// TwinCAT 3 PLC project ReleaseManager
// ProgramVersion: 3.1.4023.0
// libraries:
//   Tc2_Standard, * (Beckhoff Automation GmbH)
//   Tc2_System, * (Beckhoff Automation GmbH)
//   Tc3_Module, * (Beckhoff Automation GmbH)
// project tree:
//   / PlcTask.TcTTO
//   POUs/ MAIN.TcPOU, ReleaseClient.TcPOU, ReleaseHybrid.TcPOU, ReleaseMaster.TcPOU, TestModule_1.TcPOU, TestModule_2.TcPOU, TestModule_3.TcPOU
// real-time tasks:
//   TASK PlcTask: cycle T#10ms, priority 20, ADS port 350

CONFIGURATION ReleaseManager
    RESOURCE PLC ON TwinCAT3
        TASK PlcTask(INTERVAL := T#10ms, PRIORITY := 20);
        PROGRAM MAIN WITH PlcTask : MAIN;
    END_RESOURCE
END_CONFIGURATION

// ---- POUs/MAIN.TcPOU
PROGRAM MAIN
VAR
	fbTestModule1 : TestModule_1;
	fbTestModule2 : TestModule_2;
	fbTestModule3,fbTestModule4,fbTestModule5 : TestModule_3;
END_VAR

fbTestModule1();
fbTestModule2();

//fbTestModule1.fbNextStationReleaseClient.bReleasePresent := fbTestModule2.fbNextStationReleaseMaster.bSetRelease;
//fbTestModule2.fbNextStationReleaseMaster.bReleaseAckIn := fbTestModule1.fbNextStationReleaseClient.bReleaseAckOut;

fbTestModule2.fbNextStationReleaseMaster.SetReleaseClient(fbTestModule1.fbNextStationReleaseClient);
fbTestModule3.fbNextStationReleaseHybrid.SetReleaseClient(fbTestModule4.fbNextStationReleaseHybrid);
fbTestModule4.fbNextStationReleaseHybrid.SetReleaseClient(fbTestModule5.fbNextStationReleaseHybrid);

END_PROGRAM

// ---- POUs/TestModule_1.TcPOU
FUNCTION_BLOCK TestModule_1
VAR_INPUT
	fbNextStationReleaseClient : ReleaseClient;
END_VAR
VAR_OUTPUT
END_VAR
VAR
END_VAR

fbNextStationReleaseClient();

END_FUNCTION_BLOCK

// ---- POUs/ReleaseClient.TcPOU
FUNCTION_BLOCK ReleaseClient
VAR_INPUT
	bReleasePresent : BOOL;
END_VAR

VAR_OUTPUT
	bReleaseAckOut : BOOL;
	bLastHandshakeSuccesful : BOOL;
	bMasterAbortedLastHandshake : BOOL;
END_VAR

VAR
	fbReleasePresentEvent : R_TRIG;
	fbReleaseGoneEvent : F_TRIG;
	fbReleaseAckOutEvent : R_TRIG;
	fbReleaseAckOutGoneEvent : F_TRIG;
END_VAR

fbReleasePresentEvent(CLK:=bReleasePresent);
fbReleaseAckOutEvent(CLK:=bReleaseAckOut);
fbReleaseGoneEvent(CLK:=bReleasePresent);
fbReleaseAckOutGoneEvent(CLK:=bReleaseAckOut);

IF fbReleaseAckOutEvent.Q
THEN
	OnReleaseAckOut();
END_IF

IF fbReleasePresentEvent.Q
THEN
	OnReleasePresent();
END_IF

IF fbReleaseGoneEvent.Q
THEN
	OnReleaseGone();
END_IF

IF fbReleaseAckOutGoneEvent.Q
THEN
	OnHandshakeSuccessful();
END_IF

METHOD OnHandshakeSuccessful : BOOL
VAR_INPUT
END_VAR
bLastHandshakeSuccesful := TRUE;
END_METHOD

METHOD OnReleaseAckOut : BOOL
VAR_INPUT
END_VAR
END_METHOD

METHOD OnReleaseGone : BOOL
VAR_INPUT
END_VAR
IF bReleaseAckOut
THEN
	bReleaseAckOut := FALSE;
ELSE
	bMasterAbortedLastHandshake := TRUE;
END_IF
END_METHOD

METHOD  OnReleasePresent : BOOL
VAR_INPUT
END_VAR
bLastHandshakeSuccesful := FALSE;
bMasterAbortedLastHandshake := FALSE;
END_METHOD

END_FUNCTION_BLOCK

// ---- POUs/TestModule_2.TcPOU
FUNCTION_BLOCK TestModule_2
VAR_INPUT
	fbNextStationReleaseMaster : ReleaseMaster;
END_VAR
VAR_OUTPUT
END_VAR
VAR
END_VAR

fbNextStationReleaseMaster();

END_FUNCTION_BLOCK

// ---- POUs/ReleaseMaster.TcPOU
FUNCTION_BLOCK ReleaseMaster
VAR_INPUT
	bReleaseAckIn : BOOL;
END_VAR

VAR_OUTPUT
	bSetRelease : BOOL;
	bLastHandshakeSuccesful : BOOL;
END_VAR


VAR
	fbReleaseAckInEvent : R_TRIG;
	fbSetReleaseEvent : R_TRIG;
	fbHandshakeSuccessfulEvent : R_TRIG;
END_VAR

fbReleaseAckInEvent(CLK:=bReleaseAckIn);
fbSetReleaseEvent(CLK:=bSetRelease);

IF fbReleaseAckInEvent.Q
THEN
	OnReleaseAckIn();
END_IF

IF fbSetReleaseEvent.Q
THEN
	OnSetRelease();
END_IF

IF fbHandshakeSuccessfulEvent.Q
THEN	
	OnHandshakeSuccessful();
END_IF

METHOD OnHandshakeSuccessful : BOOL
VAR_INPUT
END_VAR
bLastHandshakeSuccesful := TRUE;
END_METHOD

METHOD OnReleaseAckIn : BOOL
VAR_INPUT
END_VAR
bSetRelease := FALSE;
END_METHOD

METHOD OnSetRelease : BOOL
VAR_INPUT
END_VAR
bLastHandshakeSuccesful := FALSE;
END_METHOD

METHOD SetReleaseClient : BOOL
VAR_IN_OUT
	fbReleaseClient : ReleaseClient;
END_VAR
bReleaseAckIn := fbReleaseClient.bReleaseAckOut;
fbReleaseClient.bReleasePresent := bSetRelease;

fbHandshakeSuccessfulEvent(CLK:=fbReleaseClient.bLastHandshakeSuccesful);
END_METHOD

END_FUNCTION_BLOCK

// ---- POUs/TestModule_3.TcPOU
FUNCTION_BLOCK TestModule_3
VAR_INPUT
	fbNextStationReleaseHybrid : ReleaseHybrid;
END_VAR
VAR_OUTPUT
END_VAR
VAR
END_VAR

fbNextStationReleaseHybrid();

END_FUNCTION_BLOCK

// ---- POUs/ReleaseHybrid.TcPOU
FUNCTION_BLOCK ReleaseHybrid EXTENDS ReleaseClient
VAR_INPUT
	bReleaseAckIn : BOOL;
END_VAR

VAR_OUTPUT
	bSetRelease : BOOL;
	bLastHandshakeSuccesfulHybrid : BOOL;
END_VAR


VAR
	fbReleaseAckInEvent : R_TRIG;
	fbSetReleaseEvent : R_TRIG;
	fbHandshakeSuccessfulEvent : R_TRIG;
END_VAR

SUPER^();
fbReleaseAckInEvent(CLK:=bReleaseAckIn);
fbSetReleaseEvent(CLK:=bSetRelease);

IF fbReleaseAckInEvent.Q
THEN
	OnReleaseAckIn();
END_IF

IF fbSetReleaseEvent.Q
THEN
	OnSetRelease();
END_IF

IF fbHandshakeSuccessfulEvent.Q
THEN	
	bLastHandshakeSuccesful := TRUE;
END_IF

METHOD OnHandshakeSuccessful : BOOL
VAR_INPUT
END_VAR
END_METHOD

METHOD OnReleaseAckIn : BOOL
VAR_INPUT
END_VAR
bSetRelease := FALSE;
END_METHOD

METHOD OnSetRelease : BOOL
VAR_INPUT
END_VAR
bLastHandshakeSuccesfulHybrid := FALSE;
END_METHOD

METHOD SetReleaseClient : BOOL
VAR_IN_OUT
	fbReleaseClient : ReleaseClient;
END_VAR
bReleaseAckIn := fbReleaseClient.bReleaseAckOut;
fbReleaseClient.bReleasePresent := bSetRelease;

fbHandshakeSuccessfulEvent(CLK:=fbReleaseClient.bLastHandshakeSuccesful);
END_METHOD

END_FUNCTION_BLOCK
